// TIA Portal project "TIAv15_Industrial_Gateway" (V15)
// My Thesis

(* hardware
DEVICE "S7-1200 station_1"  S7-1200 Station
   slot 0: "Rack_0"  S7-1200 Rack  Rack  V1.0
   slot 1: "PLC_1"  CPU 1214C DC/DC/DC  6ES7 214-1AG31-0XB0  V3.0
*)

// ===== PLC "PLC_1"  CPU 1214C DC/DC/DC =====

VAR_GLOBAL   // PLC tag table "Default tag table"
   "Clock_Byte" AT %MB0 : Byte;
   "Clock_10Hz" AT %M0.0 : Bool;
   "Clock_5Hz" AT %M0.1 : Bool;
   "Clock_2.5Hz" AT %M0.2 : Bool;
   "Clock_2Hz" AT %M0.3 : Bool;
   "Clock_1.25Hz" AT %M0.4 : Bool;
   "Clock_1Hz" AT %M0.5 : Bool;
   "Clock_0.625Hz" AT %M0.6 : Bool;
   "Clock_0.5Hz" AT %M0.7 : Bool;
   "CTU_1_R" AT %M1.0 : Bool;
END_VAR

VAR_GLOBAL   // PLC tag table "HOLD_REG"
   "40001" AT %MW100 : Word;
   "40002" AT %MW102 : Word;
   "40003" AT %MW104 : Word;
   "40004" AT %MW106 : Word;
   "40005" AT %MW108 : Word;
   "40006" AT %MW110 : Word;
   "40007" AT %MW112 : Word;
   "40008" AT %MW114 : Word;
   "40009" AT %MW116 : Word;
   "40010" AT %MW118 : Word;
   "40011" AT %MW120 : Word;
   "40012" AT %MW122 : Word;
   "40013" AT %MW124 : Word;
   "40014" AT %MW126 : Word;
   "40015" AT %MW128 : Word;
   "40016" AT %MW130 : Word;
   "40017" AT %MW132 : Word;
   "40018" AT %MW134 : Word;
   "40019" AT %MW136 : Word;
   "40020" AT %MW138 : Word;
END_VAR

DATA_BLOCK "MB_Server_Data"   // DB2
{ S7_Optimized_Access := 'TRUE' }
VERSION : 0.1
   VAR
      CONNECT_ID : UInt := 2;
      IP_PORT : UInt := 502;
      NDR : Bool;
      DR : Bool;
      ERROR : Bool;
      STATUS : Word;
   END_VAR
BEGIN
END_DATA_BLOCK

DATA_BLOCK "MB_Client_Data"   // DB5
{ S7_Optimized_Access := 'TRUE' }
VERSION : 0.1
   VAR
      DISCONNECT : Bool;
      CONNECT_ID : UInt := 1;
      IP_ADDRESS : Array[0..3] of Byte;
      IP_PORT : UInt := 502;
      MB_MODE : USInt := 1;
      DATA_ADDRESS : UDInt := 0;
      DATA_LEN : UInt := 20;
      DONE : Bool;
      BUSY : Bool;
      ERROR : Bool;
      STATUS : Word;
   END_VAR
BEGIN
   IP_ADDRESS[0] := 192;
   IP_ADDRESS[1] := 168;
   IP_ADDRESS[2] := 0;
   IP_ADDRESS[3] := 103;
END_DATA_BLOCK

DATA_BLOCK "MB_CLient_Buff"   // DB6
{ S7_Optimized_Access := 'FALSE' }
VERSION : 0.1
   VAR
      DATA : Array[0..19] of Word;
   END_VAR
BEGIN
END_DATA_BLOCK

ORGANIZATION_BLOCK "Main"   // OB1, LAD, ProgramCycle
TITLE = "Main Program Sweep (Cycle)"
{ S7_Optimized_Access := 'TRUE' }
VERSION : 0.1
BEGIN

REGION Network 1
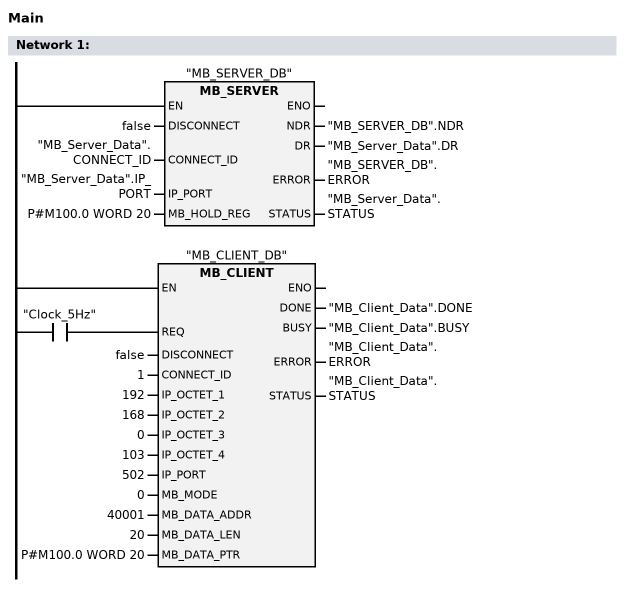
   "MB_SERVER_DB"(DISCONNECT := false,   // MB_SERVER
                  CONNECT_ID := "MB_Server_Data".CONNECT_ID,
                  IP_PORT := "MB_Server_Data".IP_PORT,
                  MB_HOLD_REG := P#M100.0 WORD 20,
                  NDR => "MB_SERVER_DB".NDR,
                  DR => "MB_Server_Data".DR,
                  ERROR => "MB_SERVER_DB".ERROR,
                  STATUS => "MB_Server_Data".STATUS);
   "MB_CLIENT_DB"(REQ := "Clock_5Hz",   // MB_CLIENT
                  DISCONNECT := false,
                  CONNECT_ID := 1,
                  IP_OCTET_1 := 192,
                  IP_OCTET_2 := 168,
                  IP_OCTET_3 := 0,
                  IP_OCTET_4 := 103,
                  IP_PORT := 502,
                  MB_MODE := 0,
                  MB_DATA_ADDR := 40001,
                  MB_DATA_LEN := 20,
                  MB_DATA_PTR := P#M100.0 WORD 20,
                  DONE => "MB_Client_Data".DONE,
                  BUSY => "MB_Client_Data".BUSY,
                  ERROR => "MB_Client_Data".ERROR,
                  STATUS => "MB_Client_Data".STATUS);
END_REGION
END_ORGANIZATION_BLOCK